PROGRAM NorthLight_Control
VAR
	StraightGreenLight  : BOOL := FALSE;	//Controls if the green light is on
	StraightYellowLight : BOOL := FALSE;	//Controls if the yellow light is on
	StraightRedLight    : BOOL := TRUE; 	//Controls if the red light is on
	
	StraightOnTimer : INT := 0;				//Tracks how long the light has been on
	
	LeftGreenLight  : BOOL := FALSE;		//Controls if the green light is on
	LeftYellowLight : BOOL := FALSE;		//Controls if the yellow light is on
	leftRedLight    : BOOL := TRUE; 		//Controls if the red light is on
	
	LeftOnTimer : INT := 0;					//Tracks how long the light has been on
	
	CrosswalkLight : BOOL := FALSE;			//Controls if the crosswalk light is on (walk=TRUE)
END_VAR

//If all of the sensors and lights are off, default to N/S straight
IF Glbl.northStraightSensor = FALSE AND  Glbl.northLeftSensor = FALSE AND Glbl.southStraightSensor = FALSE AND Glbl.southLeftSensor = FALSE AND Glbl.eastStraightSensor = FALSE AND Glbl.eastLeftSensor = FALSE AND Glbl.westStraightSensor = FALSE AND Glbl.westLeftSensor = FALSE AND  Glbl.northLeftActive = FALSE AND Glbl.southLeftActive = FALSE AND Glbl.eastStraightActive = FALSE AND Glbl.eastLeftActive = FALSE AND Glbl.westStraightActive = FALSE AND Glbl.westLeftActive = FALSE THEN
	Glbl.northStraightActive := TRUE;
	StraightRedLight := FALSE;
	StraightGreenLight := TRUE;
	Glbl.state1Counter := 0;
	Glbl.state2Counter := 0;
	Glbl.state3Counter := 0;
	Glbl.state4Counter := 0;
	Glbl.state5Counter := 0;
	Glbl.state6Counter := 0;
	Glbl.state7Counter := 0;
	Glbl.state8Counter := 0;
	
ELSE//Control for the straight light if active
	IF Glbl.northStraightActive = TRUE THEN			//If the straight light is set to be active
		IF StraightOnTimer = 0 THEN					//Take off half of the state counter when the light is activated
			//Glbl.state1Counter := Glbl.state1Counter - (Glbl.state1Counter/2);
			//Glbl.state5Counter := Glbl.state5Counter - (Glbl.state5Counter/2);		
		END_IF
		IF StraightOnTimer <= 10 THEN				//If the light has been on for 10 seconds or less, make it green
			StraightGreenLight := TRUE;
			StraightYellowLight := FALSE;
			StraightRedLight := FALSE;
			StraightOnTimer := StraightOnTimer + 1;	//Incriment the amount of time it has been on by 1
			Glbl.northStraightSensor := FALSE;		//Set the sensor to false
			Glbl.northStraightSensorCnt := MAX(Glbl.northStraightSensorCnt-1, 0);		//Set the car counter to 0
		ELSIF StraightOnTimer <= 13 THEN			//If the light has been on for 11-13 seconds, make it yellow
			StraightGreenLight := FALSE;
			StraightYellowLight := TRUE;
			StraightRedLight := FALSE;
			StraightOnTimer := StraightOnTimer + 1;	//Incriment the amount of time it has been on by 1
		ELSE										//Once it is done, turn it to red and set it as inactive, reset timer to 0
			StraightGreenLight := FALSE;
			StraightYellowLight := FALSE;
			StraightRedLight := TRUE;
			Glbl.northStraightActive := FALSE;
			StraightOnTimer := 0;	
		END_IF
	END_IF
END_IF

//Control for the left light if active
IF Glbl.northLeftActive = TRUE THEN			//If the left light is set to be active
	IF LeftOnTimer = 0 THEN					//Take off half of the state counter when the light is activated
		//Glbl.state3Counter := Glbl.state3Counter - (Glbl.state3Counter/2);
		//Glbl.state5Counter := Glbl.state5Counter - (Glbl.state5Counter/2);	
	END_IF
	IF LeftOnTimer <= 10 THEN				//If the light has been on for 10 seconds or less, make it green
		LeftGreenLight := TRUE;
		LeftYellowLight := FALSE;
		LeftRedLight := FALSE;
		LeftOnTimer := LeftOnTimer + 1;	//Incriment the amount of time it has been on by 1
		Glbl.northLeftSensor := FALSE; 		//Set the sensor to false
		Glbl.northLeftSensorCnt := MAX(Glbl.northLeftSensorCnt-1, 0);
	ELSIF LeftOnTimer <= 13 THEN			//If the light has been on for 11-13 seconds, make it yellow
		LeftGreenLight := FALSE;
		LeftYellowLight := TRUE;
		LeftRedLight := FALSE;
		LeftOnTimer := LeftOnTimer + 1;	//Incriment the amount of time it has been on by 1
	ELSE									//Once it is done, turn it to red and set it as inactive, reset timer to 0
		LeftGreenLight := FALSE;
		LeftYellowLight := FALSE;
		LeftRedLight := TRUE;
		Glbl.northLeftActive := FALSE;
		LeftOnTimer := 0;	
	END_IF
END_IF

//If the sensor is on and the light is off, incirment the waiting counters
IF Glbl.northStraightSensor = TRUE AND Glbl.northStraightActive = FALSE THEN
	Glbl.state1Counter := Glbl.state1Counter + Glbl.northStraightSensorCnt;
	Glbl.state5Counter := Glbl.state5Counter + Glbl.northStraightSensorCnt;
END_IF
IF Glbl.northLeftSensor = TRUE AND Glbl.northLeftActive = FALSE THEN
	Glbl.state3Counter := Glbl.state3Counter + Glbl.northLeftSensorCnt;
	Glbl.state5Counter := Glbl.state5Counter + Glbl.northLeftSensorCnt;
END_IF

//Check to see if the crosswalk can be turned on
IF (Glbl.eastStraightActive = TRUE AND Glbl.westStraightActive = TRUE) OR (Glbl.eastStraightActive = TRUE AND Glbl.eastLeftActive = TRUE) THEN
	CrosswalkLight := TRUE;
ELSE
	CrosswalkLight := FALSE;
END_IF

END_PROGRAM

(* stored: Version 1.1.0.1, ProductVersion 3.1.4022.10
   POU NorthLight_Control: Id {934537e3-63a4-40c0-986a-6c025fb28c9d}, SpecialFunc None *)
